PROGRAM MAIN
VAR
	InitComplete: BOOL;
	
	//Function Block INIT
	FB_hmi_connection: FB_hmi_connection;
	FB_WindingControl: FB_WindingControl;
	FB_EventLogger: FB_EventLogger;
	FB_FileReadWrite: FB_fileReadWrite;
	
	
	
	
	
END_VAR

CYCLIC();

METHOD CYCLIC : BOOL
VAR_INPUT
END_VAR
IF NOT InitComplete THEN
    InitComplete := INIT();
    RETURN;
END_IF

//FB Cyclic logic. 

FB_EventLogger.CYCLIC(); //event logger
FB_hmi_connection.CYCLIC(); //hmi inputs and outputs
FB_WindingControl.CYCLIC(); //motor control. 
FB_FileReadWrite.CYLIC();
END_METHOD

METHOD INIT : BOOL
VAR_INPUT
END_VAR
//Function Block INIT
FB_hmi_connection.INIT();
FB_WindingControl.INIT();
FB_EventLogger.INIT();
//MAIN INIT


FB_WindingControl.hmiConnection:=ADR(FB_hmi_connection);
FB_WindingControl.eventLogger:=ADR(FB_EventLogger);
FB_WindingControl.fileReadWrite:=ADR(FB_fileReadWrite);

INIT:=TRUE;
END_METHOD

END_PROGRAM

(* stored: Version 1.1.0.1, ProductVersion 3.1.4024.12
   POU MAIN: Id {89db02fc-403c-41e5-9629-9f906630e622}, SpecialFunc None
   Folder Methods: Id {5be72f40-ae86-44c7-98c0-16546f0605de}
   Folder Init Methods: Id {56da2c24-90a7-4142-9494-8c615ded5ee6}
   Method CYCLIC: Id {18bc88a2-8c6d-4614-9e8b-5364e5c9f027}
   Method INIT: Id {d283a7a7-3eaa-4933-86d8-aab52f7a452a} *)
